TYPE ST_RemoveReservationData :
STRUCT
	sObjectID					: STRING := 'MAIN.fbMMServer';
	sMethodID					: STRING := 'MAIN.fbMMServer#M_RemoveReservationList';
	iStatus						: INT;
	iNoOfInputArgs				: BYTE := 2;
	iNoOfOutputArgs				: BYTE := 2;
	stInput						: ST_RemoveReservationDataIn;
	stOutput					: ST_RemoveReservationDataOut;	
END_STRUCT
END_TYPE

(* stored: Version 1.1.0.1, ProductVersion 3.1.4024.5
   DUT ST_RemoveReservationData: Id {21aa7295-838d-4f35-a51c-b8211b05cad9} *)
